# EPICS substitutions: iocTops/EdwardsNextTurbo-2-4/iocs/example_EdwardsNextTurbo/example_EdwardsNextTurboApp/Db/example_EdwardsNextTurbo.substitutions
file EdwardsNextTurbo.template
{
pattern { P, port }
{ TS-VA-TURBO-01, TS-VA-TURBO-01 }
}
